% RSLogix 500 project PID-Substitution-Logic.RSS, saved by version 8.30.00.16 %
PROJECT "UNTITLED"    % processor: Bul.1763 MicroLogix 1100 Series B %

PROGRAM FILES
  LAD 2   10 rungs

DATA FILES
  O0 OUTPUT  4 elements
  I1 INPUT  6 elements
  S2 STATUS  66 elements
  B3 BINARY  1 elements
  T4 TIMER  1 elements
  C5 COUNTER  1 elements
  R6 CONTROL  1 elements
  N7 INTEGER  15 elements
  F8 FLOAT  1 elements

LADDER 2
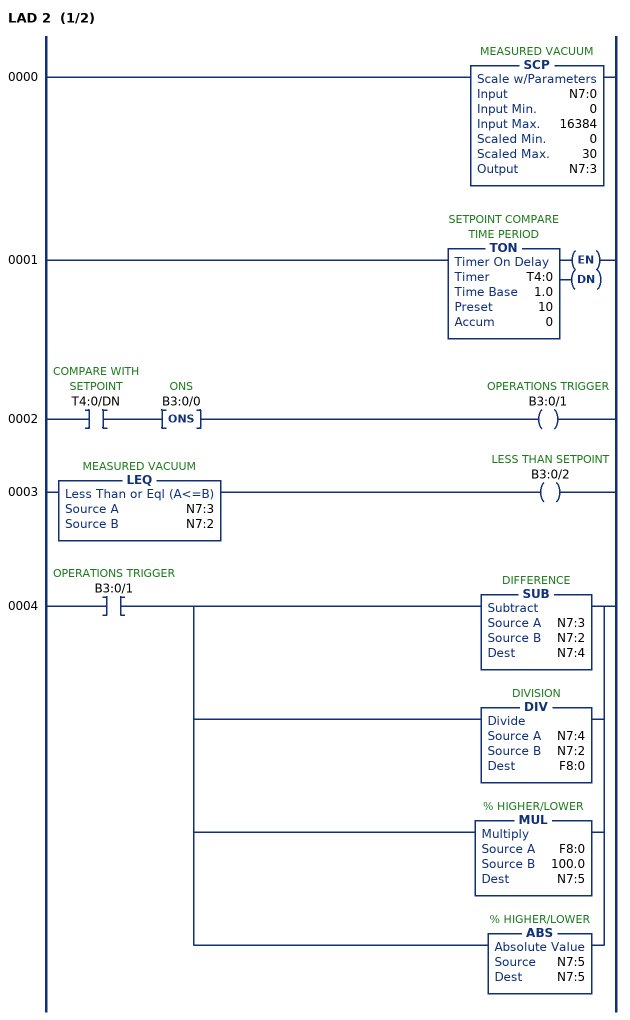
% Rung: 0 %
SOR SCP N7:0 0 16384 0 30 N7:3 EOR
%   N7:0  "VACUUM SENSOR IN" %
%   N7:3  "MEASURED VACUUM" %
% Rung: 1 %
SOR TON T4:0 1.0 10 0 EOR
%   T4:0  "SETPOINT COMPARE TIME PERIOD" %
% Rung: 2 %
SOR XIC T4:0/DN ONS B3:0/0 OTE B3:0/1 EOR
%   T4:0/DN  "COMPARE WITH SETPOINT" %
%   B3:0/0  "ONS" %
%   B3:0/1  "OPERATIONS TRIGGER" %
% Rung: 3 %
SOR LEQ N7:3 N7:2 OTE B3:0/2 EOR
%   N7:3  "MEASURED VACUUM" %
%   N7:2  "VACUUM SETPOINT" %
%   B3:0/2  "LESS THAN SETPOINT" %
% Rung: 4 %
SOR XIC B3:0/1 BST SUB N7:3 N7:2 N7:4 NXB DIV N7:4 N7:2 F8:0 NXB MUL F8:0 100.0 N7:5 NXB ABS N7:5 N7:5 BND EOR
%   B3:0/1  "OPERATIONS TRIGGER" %
%   N7:3  "MEASURED VACUUM" %
%   N7:2  "VACUUM SETPOINT" %
%   N7:4  "DIFFERENCE" %
%   F8:0  "DIVISION" %
%   N7:5  "% HIGHER/LOWER" %

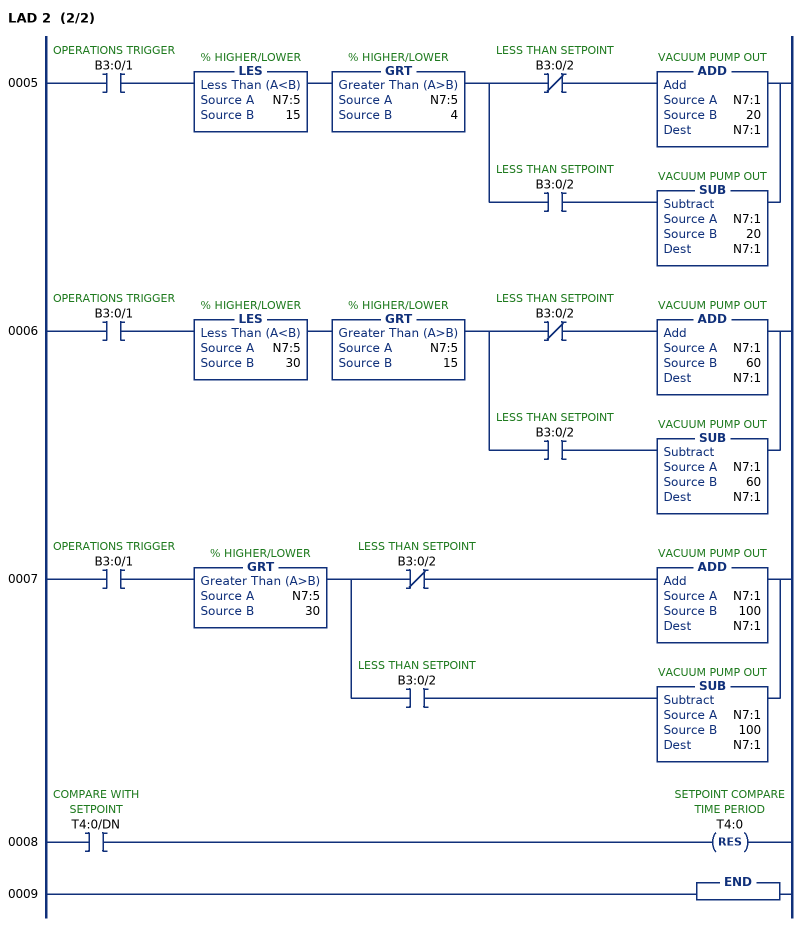
% Rung: 5 %
SOR XIC B3:0/1 LES N7:5 15 GRT N7:5 4 BST XIO B3:0/2 ADD N7:1 20 N7:1 NXB XIC B3:0/2 SUB N7:1 20 N7:1 BND EOR
%   B3:0/1  "OPERATIONS TRIGGER" %
%   N7:5  "% HIGHER/LOWER" %
%   B3:0/2  "LESS THAN SETPOINT" %
%   N7:1  "VACUUM PUMP OUT" %
% Rung: 6 %
SOR XIC B3:0/1 LES N7:5 30 GRT N7:5 15 BST XIO B3:0/2 ADD N7:1 60 N7:1 NXB XIC B3:0/2 SUB N7:1 60 N7:1 BND EOR
%   B3:0/1  "OPERATIONS TRIGGER" %
%   N7:5  "% HIGHER/LOWER" %
%   B3:0/2  "LESS THAN SETPOINT" %
%   N7:1  "VACUUM PUMP OUT" %
% Rung: 7 %
SOR XIC B3:0/1 GRT N7:5 30 BST XIO B3:0/2 ADD N7:1 100 N7:1 NXB XIC B3:0/2 SUB N7:1 100 N7:1 BND EOR
%   B3:0/1  "OPERATIONS TRIGGER" %
%   N7:5  "% HIGHER/LOWER" %
%   B3:0/2  "LESS THAN SETPOINT" %
%   N7:1  "VACUUM PUMP OUT" %
% Rung: 8 %
SOR XIC T4:0/DN RES T4:0 EOR
%   T4:0/DN  "COMPARE WITH SETPOINT" %
%   T4:0  "SETPOINT COMPARE TIME PERIOD" %
% Rung: 9 %
SOR END EOR

DATA TABLE (non-zero values as saved)
DATA T4
% .PRE .ACC %
% T4:0 % 10 0
DATA N7
% N7:0 % 8192 6000 15 0 0 0 0 0 0 0
